FUNCTION_BLOCK CheckWatchdog
VAR_INPUT
	EN: BOOL;
	Watchdog: INT;
	Timeout: TIME := T#30S;
END_VAR
VAR_OUTPUT
	ENO: BOOL;
	Alarm: BOOL;
END_VAR
VAR
	LastWatchdog: INT;
	WatchdogTimer: Timer;
	FirstTime: bool;
END_VAR

IF NOT FirstTime THEN
	WatchdogTimer.Restart();
	FirstTime := TRUE;
END_IF
ENO := EN;
IF EN THEN
	IF Watchdog <> LastWatchdog THEN
		WatchdogTimer.Restart();	
		LastWatchdog := Watchdog;
	END_IF
	Alarm := WatchdogTimer.ElapsedTime() > TO_LINT(Timeout);
ELSE
	WatchdogTimer.Restart();	
	Alarm := FALSE;
END_IF

END_FUNCTION_BLOCK

(* stored: Version 1.1.0.1, ProductVersion 3.1.4024.6
   POU CheckWatchdog: Id {1cabb147-68a0-4ddd-84b0-c821a7f35d4a}, SpecialFunc None *)
